(* PLC project benzene-distillation, Generated TextualNotationConverter 1.0 *)
(* stored: creationDateTime 2025-07-30T12:00:00, modificationDateTime 2025-01-30T12:00:00 *)

FUNCTION_BLOCK ANALOG_IN
  VAR_INPUT
    Name : STRING;
    Description : STRING;
    Raw_Signal : REAL;
    PV_High : REAL;
    PV_Low : REAL;
    Scaling_Slope : REAL;
    Scaling_Offset : REAL;
    Alarm_Enable : BOOL;
  END_VAR
  VAR_OUTPUT
    PV : REAL;
    High_Alarm : BOOL;
    Low_Alarm : BOOL;
    General_Fault : BOOL;
  END_VAR

            
          
END_FUNCTION_BLOCK

FUNCTION_BLOCK DIGITAL_IN
  VAR_INPUT
    Name : STRING;
    Description : STRING;
    DI_Raw : BOOL;
    DebounceTime : STRING;
    EnableAlarm : BOOL;
  END_VAR
  VAR_OUTPUT
    DI_Out : BOOL;
    Fault_State : BOOL;
  END_VAR

            
          
END_FUNCTION_BLOCK

FUNCTION_BLOCK PID_BASIC
  VAR_INPUT
    Name : STRING;
    Description : STRING;
    AUTO : BOOL;
    PV : REAL;
    SP : REAL;
    MV_MIN : REAL;
    MV_MAX : REAL;
    X0 : REAL;
    KP : REAL;
    TR : REAL;
    TD : REAL;
    PV_High : REAL;
    PV_Low : REAL;
    Deviation_Limit : REAL;
    Inhibit : BOOL;
  END_VAR
  VAR_OUTPUT
    PV_High_Alarm : BOOL;
    PV_Low_Alarm : BOOL;
    Deviation_Alarm : BOOL;
    XOUT : REAL;
  END_VAR

            
          
END_FUNCTION_BLOCK

FUNCTION_BLOCK VALVE_ELECTRIC
  VAR_INPUT
    Name : STRING;
    Description : STRING;
    Control_Signal : REAL;
    Manual_Mode : BOOL;
    Manual_Position : REAL;
    Open_Limit : REAL;
    Close_Limit : REAL;
    Timeout : STRING;
    Inhibit : BOOL;
  END_VAR
  VAR_OUTPUT
    Valve_Position : REAL;
    Feedback_Pos : REAL;
    Valve_Moving : BOOL;
    Position_Error : BOOL;
    Alarm : BOOL;
  END_VAR

            
          
END_FUNCTION_BLOCK

FUNCTION_BLOCK VALVE_ON_OFF
  VAR_INPUT
    Name : STRING;
    Description : STRING;
    Open_Cmd : BOOL;
    Close_Cmd : BOOL;
    Timeout : STRING;
    Inhibit : BOOL;
  END_VAR
  VAR_OUTPUT
    FB_Opened : BOOL;
    FB_Closed : BOOL;
    Valve_Open_Out : BOOL;
    Valve_Close_Out : BOOL;
    Alarm_Position_Error : BOOL;
    Alarm_General : BOOL;
  END_VAR

            
          
END_FUNCTION_BLOCK

PROGRAM Section2
  VAR
    TE101_BaseTemp_PV : REAL;
    PV103_MV_Command : REAL;
    PV103_Position_Feedback : REAL;
    XV105_Open_Feedback : BOOL;
    LIT101_ColumnLevel_PV : REAL;
    PIT102_Pressure_PV : REAL;
  END_VAR
  VAR
    TE-101 : ANALOG_IN;
    TIC-104 : PID_BASIC;
    PV-103 : VALVE_ELECTRIC;
    XV-105 : VALVE_ON_OFF;
    LIT-101 : ANALOG_IN;
    PIT-102 : ANALOG_IN;
    LAH-101 : DIGITAL_IN;
    LAL-101 : DIGITAL_IN;
  END_VAR
  VAR  (* added by the conversion: wires and edge detectors of the diagram *)
    _OR1_OUT : BOOL;
  END_VAR

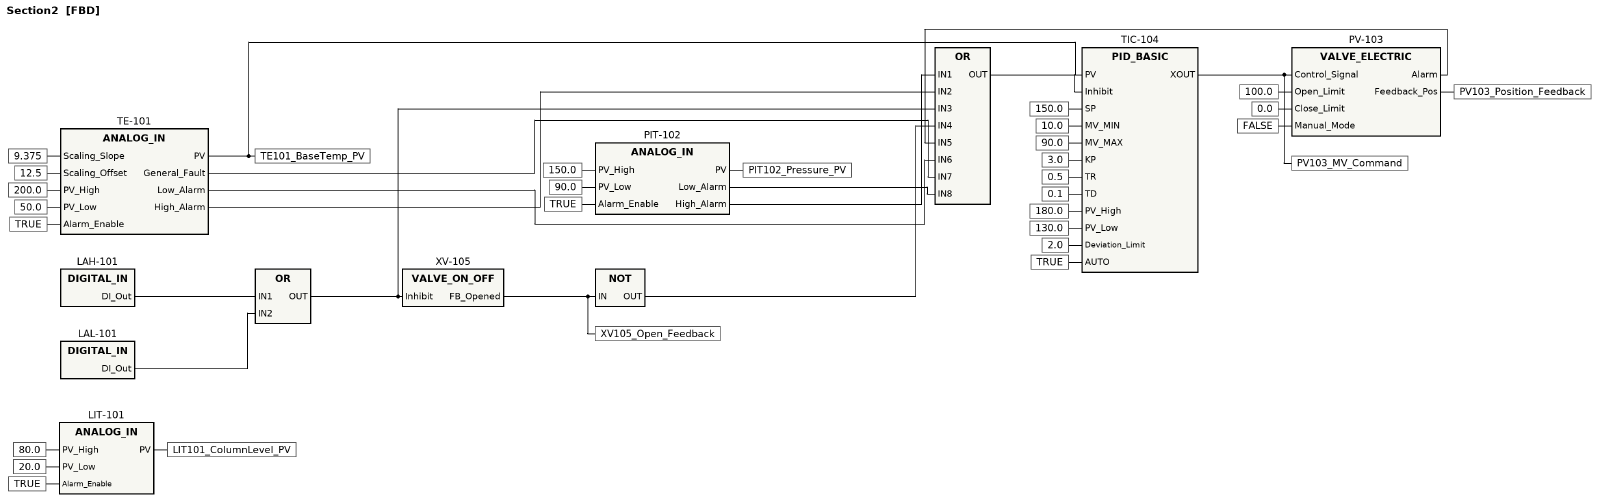
(* FBD diagram, written out as Structured Text *)
LIT-101(PV_High := 80.0, PV_Low := 20.0, Alarm_Enable := TRUE);
LIT101_ColumnLevel_PV := LIT-101.PV;
PIT-102(PV_High := 150.0, PV_Low := 90.0, Alarm_Enable := TRUE);
PIT102_Pressure_PV := PIT-102.PV;
TE-101(Scaling_Slope := 9.375, Scaling_Offset := 12.5, PV_High := 200.0, PV_Low := 50.0, Alarm_Enable := TRUE);
LAH-101();
LAL-101();
_OR1_OUT := LAH-101.DI_Out OR LAL-101.DI_Out;
XV-105(Inhibit := _OR1_OUT);
PV-103(Control_Signal := TIC-104.XOUT, Open_Limit := 100.0, Close_Limit := 0.0, Manual_Mode := FALSE);
TIC-104(PV := TE-101.PV, Inhibit := PIT-102.High_Alarm OR TE-101.High_Alarm OR _OR1_OUT OR NOT XV-105.FB_Opened OR PV-103.Alarm OR TE-101.Low_Alarm OR TE-101.General_Fault OR PIT-102.Low_Alarm, SP := 150.0, MV_MIN := 10.0, MV_MAX := 90.0, KP := 3.0, TR := 0.5, TD := 0.1, PV_High := 180.0, PV_Low := 130.0, Deviation_Limit := 2.0, AUTO := TRUE);
PV103_MV_Command := TIC-104.XOUT;
PV103_Position_Feedback := PV-103.Feedback_Pos;
TE101_BaseTemp_PV := TE-101.PV;
XV105_Open_Feedback := XV-105.FB_Opened;
END_PROGRAM

FUNCTION_BLOCK BOOL_IN
  VAR_INPUT
    Name : STRING;
    Description : STRING;
    Bool_In : BOOL;
    Alarm_OnTrue : BOOL;
    Alarm_OnFalse : BOOL;
    Latch_Enable : BOOL;
    Reset_Latch : BOOL;
  END_VAR
  VAR_OUTPUT
    Bool_Out : BOOL;
    Alarm_Active : BOOL;
    Latched_Status : BOOL;
  END_VAR

            
          
END_FUNCTION_BLOCK

FUNCTION_BLOCK DUTY_STANDBY
  VAR_INPUT
    Name : STRING;
    Description : STRING;
    Enable : BOOL;
    StartRequest : BOOL;
    AlternateEnable : BOOL;
    ForcePumpA : BOOL;
    ForcePumpB : BOOL;
    DutyElapsed : BOOL;
    MinRunElapsed : BOOL;
    SwitchoverDelayElapsed : BOOL;
    StartTimeoutElapsed : BOOL;
    PumpA_RunFB : BOOL;
    PumpB_RunFB : BOOL;
    PumpA_Fault : BOOL;
    PumpB_Fault : BOOL;
    Reset : BOOL;
    Inhibit : BOOL;
  END_VAR
  VAR_OUTPUT
    CmdPumpA : BOOL;
    CmdPumpB : BOOL;
    ActiveIsA : BOOL;
    SwitchedDueToDuty : BOOL;
    SwitchedDueToFailure : BOOL;
    Alarm_FailedStart_A : BOOL;
    Alarm_FailedStart_B : BOOL;
    Alarm_NoAvailablePump : BOOL;
  END_VAR

            
          
END_FUNCTION_BLOCK

FUNCTION_BLOCK MOTOR_2SPD
  VAR_INPUT
    Name : STRING;
    Description : STRING;
    Start_Cmd : BOOL;
    Stop_Cmd : BOOL;
    Speed_High_Cmd : BOOL;
    Speed_Low_Cmd : BOOL;
    Inhibit : BOOL;
  END_VAR
  VAR_OUTPUT
    Motor_Start_Out : BOOL;
    FB_Running : BOOL;
    FB_Trip : BOOL;
    FB_HighSpeed : BOOL;
    FB_LowSpeed : BOOL;
    Alarm_Speed_Error : BOOL;
  END_VAR

            
          
END_FUNCTION_BLOCK

FUNCTION_BLOCK MOTOR_ON_OFF
  VAR_INPUT
    Name : STRING;
    Description : STRING;
    Start_Cmd : BOOL;
    Stop_Cmd : BOOL;
    Start_Delay : STRING;
    MinRunTime : STRING;
    Inhibit : BOOL;
  END_VAR
  VAR_OUTPUT
    Motor_Start_Out : BOOL;
    FB_Running : BOOL;
    FB_Trip : BOOL;
    Alarm_Start_Fail : BOOL;
    Alarm_Stop_Fail : BOOL;
  END_VAR

            
          
END_FUNCTION_BLOCK

FUNCTION_BLOCK MOTOR_VSD
  VAR_INPUT
    Name : STRING;
    Description : STRING;
    Start_Cmd : BOOL;
    Stop_Cmd : BOOL;
    Speed_SP : REAL;
    Accel_Ramp : STRING;
    Decel_Ramp : STRING;
    Inhibit : BOOL;
  END_VAR
  VAR_OUTPUT
    Speed_Out : REAL;
    FB_Running : BOOL;
    FB_Fault : BOOL;
    FB_Ready : BOOL;
    FB_ActualSpeed : REAL;
    Alarm_Speed_Deviation : BOOL;
    Alarm_Comm_Fail : BOOL;
  END_VAR

            
          
END_FUNCTION_BLOCK

FUNCTION_BLOCK RATIO_CONTROL
  VAR_INPUT
    Name : STRING;
    Description : STRING;
    Auto : BOOL;
    PrimaryPV : REAL;
    SecondaryPV : REAL;
    RatioSP : REAL;
    Bias : REAL;
    TrimKp : REAL;
    TrimTi : STRING;
    MV_MIN : REAL;
    MV_MAX : REAL;
    ManOut : REAL;
    Inhibit : BOOL;
  END_VAR
  VAR_OUTPUT
    SlaveSP : REAL;
    ActiveRatio : REAL;
    RatioErr : REAL;
  END_VAR

            
          
END_FUNCTION_BLOCK

FUNCTION_BLOCK SPLIT_RANGE
  VAR_INPUT
    Name : STRING;
    Description : STRING;
    IN : REAL;
    Split_Point : REAL;
    Output1_Start : REAL;
    Output1_End : REAL;
    Output2_Start : REAL;
    Output2_End : REAL;
  END_VAR
  VAR_OUTPUT
    OUT1 : REAL;
    OUT2 : REAL;
  END_VAR

            
          
END_FUNCTION_BLOCK

FUNCTION_BLOCK VOTING_ANALOG
  VAR_INPUT
    Name : STRING;
    Description : STRING;
    Input1 : REAL;
    Input2 : REAL;
    Input3 : REAL;
    Deviation_Limit : REAL;
    Voting_Scheme : STRING;
    EnableAlarm : BOOL;
    Inhibit : BOOL;
  END_VAR
  VAR_OUTPUT
    Voted_Output : REAL;
    Sensor1_Fault : BOOL;
    Sensor2_Fault : BOOL;
    Sensor3_Fault : BOOL;
    Alarm_Voting_Error : BOOL;
    Healthy_Sensors_Count : INT;
  END_VAR

            
          
END_FUNCTION_BLOCK

PROGRAM Section3
  VAR
    TI_106_TemperaturePV : REAL;
    FIT_101_SteamFlowPV : REAL;
    PT_101_PressurePV : REAL;
    FIC_104_MV_Percent : REAL;
    LIC_002_LowLevelTrip : BOOL;
    FAH_104_FlowFailAlarm : BOOL;
    TAH_106_Alarm : BOOL;
    TAL_106_Alarm : BOOL;
    TCV_106_Alarm : BOOL;
    TCV_106_FeedbackPos : REAL;
  END_VAR
  VAR
    TI-106 : ANALOG_IN;
    FIT-101 : ANALOG_IN;
    PT-101 : ANALOG_IN;
    FIC-104 : PID_BASIC;
    TCV-106 : VALVE_ELECTRIC;
  END_VAR
  VAR  (* added by the conversion: wires and edge detectors of the diagram *)
    _OR42_OUT : BOOL;
  END_VAR

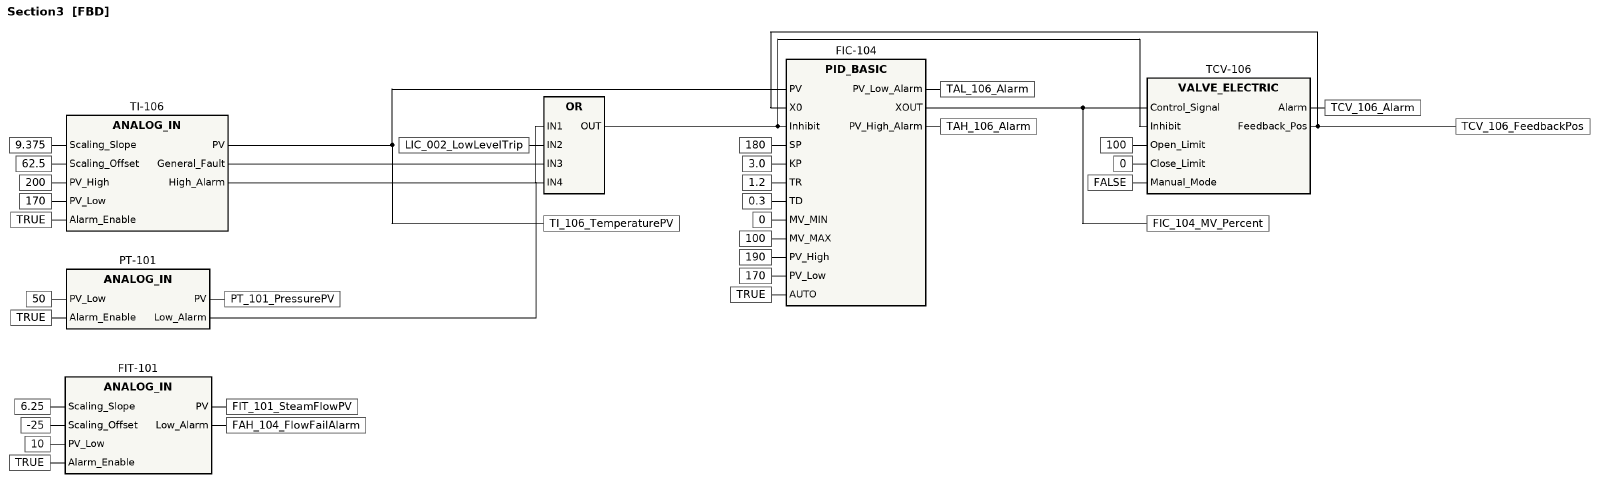
(* FBD diagram, written out as Structured Text *)
FIT-101(Scaling_Slope := 6.25, Scaling_Offset := -25, PV_Low := 10, Alarm_Enable := TRUE);
FAH_104_FlowFailAlarm := FIT-101.Low_Alarm;
TI-106(Scaling_Slope := 9.375, Scaling_Offset := 62.5, PV_High := 200, PV_Low := 170, Alarm_Enable := TRUE);
PT-101(PV_Low := 50, Alarm_Enable := TRUE);
_OR42_OUT := TI-106.High_Alarm OR LIC_002_LowLevelTrip OR TI-106.General_Fault OR PT-101.Low_Alarm;
TCV-106(Control_Signal := FIC-104.XOUT, Inhibit := _OR42_OUT, Open_Limit := 100, Close_Limit := 0, Manual_Mode := FALSE);
FIC-104(PV := TI-106.PV, X0 := TCV-106.Feedback_Pos, Inhibit := _OR42_OUT, SP := 180, KP := 3.0, TR := 1.2, TD := 0.3, MV_MIN := 0, MV_MAX := 100, PV_High := 190, PV_Low := 170, AUTO := TRUE);
FIC_104_MV_Percent := FIC-104.XOUT;
FIT_101_SteamFlowPV := FIT-101.PV;
PT_101_PressurePV := PT-101.PV;
TAH_106_Alarm := FIC-104.PV_High_Alarm;
TAL_106_Alarm := FIC-104.PV_Low_Alarm;
TCV_106_Alarm := TCV-106.Alarm;
TCV_106_FeedbackPos := TCV-106.Feedback_Pos;
TI_106_TemperaturePV := TI-106.PV;
END_PROGRAM

PROGRAM Section4
  VAR
    LT105_V104_Level_PV : REAL;
    FT107_CondensateFlow_PV : REAL;
    PT104_AccumulatorPressure_PV : REAL;
    LIC104_RSP_to_FIC107 : REAL;
    FIC107_ValveCmd_to_LV107 : REAL;
    XV103_Open_FB : BOOL;
    Cascade_Permissive_OK : BOOL;
    Startup_Delay_Done : BOOL;
  END_VAR
  VAR
    LT-105 : ANALOG_IN;
    FT-107 : ANALOG_IN;
    PT-104 : ANALOG_IN;
    LIC-104 : PID_BASIC;
    FIC-107 : PID_BASIC;
    PIC-104 : PID_BASIC;
    LV-107 : VALVE_ELECTRIC;
    XV-103 : VALVE_ON_OFF;
    LAH-104 : DIGITAL_IN;
    LAL-104 : DIGITAL_IN;
    StartupDelay : TON;
  END_VAR
  VAR  (* added by the conversion: wires and edge detectors of the diagram *)
    _OR83_OUT : BOOL;
    _NOT84_OUT : BOOL;
  END_VAR

(* FBD diagram, written out as Structured Text *)
PT-104(PV_High := 30.0, PV_Low := 15.0, Alarm_Enable := TRUE);
LT-105(PV_High := 90.0, PV_Low := 10.0, Alarm_Enable := TRUE);
XV-103();
FT-107(PV_Low := 0.0, PV_High := 50.0, Alarm_Enable := TRUE);
StartupDelay(IN := _NOT84_OUT, PT := T#30s);
LIC-104(PV := LT-105.PV, Inhibit := _OR83_OUT, AUTO := StartupDelay.Q, SP := 65.0, KP := 1.5, TR := 2.5, X0 := 40.0, MV_MIN := 0.0, MV_MAX := 100.0, PV_High := 90.0, PV_Low := 10.0);
FIC-107(SP := LIC-104.XOUT * 0.5, PV := FT-107.PV, Inhibit := _OR83_OUT, AUTO := _NOT84_OUT, KP := 4.0, TR := 0.5, MV_MIN := 0.0, MV_MAX := 100.0, X0 := 0.0);
LV-107(Control_Signal := FIC-107.XOUT, Inhibit := PT-104.High_Alarm, Manual_Mode := PT-104.High_Alarm, Manual_Position := 0.0, Close_Limit := 0.0, Open_Limit := 100.0);
_OR83_OUT := PT-104.High_Alarm OR PT-104.Low_Alarm OR LT-105.Low_Alarm OR NOT XV-103.FB_Opened OR FT-107.General_Fault OR LV-107.Position_Error;
_NOT84_OUT := NOT _OR83_OUT;
Cascade_Permissive_OK := _NOT84_OUT;
FIC107_ValveCmd_to_LV107 := FIC-107.XOUT;
FT107_CondensateFlow_PV := FT-107.PV;
LIC104_RSP_to_FIC107 := LIC-104.XOUT;
LT105_V104_Level_PV := LT-105.PV;
PT104_AccumulatorPressure_PV := PT-104.PV;
Startup_Delay_Done := StartupDelay.Q;
XV103_Open_FB := XV-103.FB_Opened;
PIC-104(PV := PT-104.PV, PV_High := 30.0, PV_Low := 15.0, MV_MIN := 0.0, MV_MAX := 100.0);
LAH-104();
LAL-104();
END_PROGRAM

PROGRAM Section5
  VAR
    FI102_FlowRate_PV : REAL;
    PI102_Pressure_PV : REAL;
    LIC102_Level_StartPermissive : BOOL;
    P102_ActiveIsA_Status : BOOL;
  END_VAR
  VAR
    FI-102 : ANALOG_IN;
    PI-102 : ANALOG_IN;
    LCV-102 : VALVE_ELECTRIC;
    LIC-102 : BOOL_IN;
    P-102A : MOTOR_ON_OFF;
    P-102B : MOTOR_ON_OFF;
    P-102 : DUTY_STANDBY;
  END_VAR
  VAR  (* added by the conversion: wires and edge detectors of the diagram *)
    _TON140_OUT : BOOL;
  END_VAR

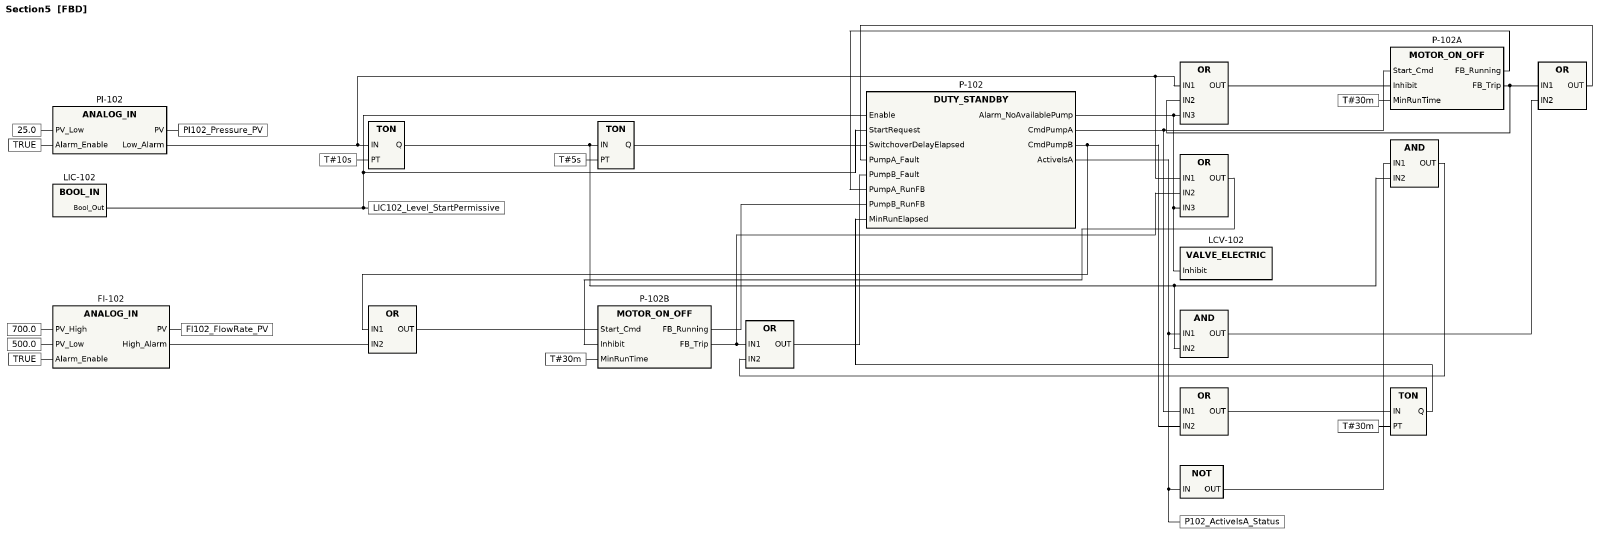
(* FBD diagram, written out as Structured Text *)
FI-102(PV_High := 700.0, PV_Low := 500.0, Alarm_Enable := TRUE);
FI102_FlowRate_PV := FI-102.PV;
LIC-102();
LIC102_Level_StartPermissive := LIC-102.Bool_Out;
PI-102(PV_Low := 25.0, Alarm_Enable := TRUE);
_TON140_OUT := TON(PI-102.Low_Alarm, T#10s);
P-102A(Start_Cmd := P-102.CmdPumpA, Inhibit := PI-102.Low_Alarm OR P-102A.FB_Trip OR P-102.Alarm_NoAvailablePump, MinRunTime := T#30m);
P-102B(Start_Cmd := P-102.CmdPumpB OR FI-102.High_Alarm, Inhibit := PI-102.Low_Alarm OR P-102B.FB_Trip OR P-102.Alarm_NoAvailablePump, MinRunTime := T#30m);
P-102(Enable := LIC-102.Bool_Out, StartRequest := LIC-102.Bool_Out, SwitchoverDelayElapsed := TON(_TON140_OUT, T#5s), PumpA_Fault := P-102A.FB_Trip OR P-102.ActiveIsA AND _TON140_OUT, PumpB_Fault := P-102B.FB_Trip OR NOT P-102.ActiveIsA AND _TON140_OUT, PumpA_RunFB := P-102A.FB_Running, PumpB_RunFB := P-102B.FB_Running, MinRunElapsed := TON(P-102.CmdPumpA OR P-102.CmdPumpB, T#30m));
P102_ActiveIsA_Status := P-102.ActiveIsA;
PI102_Pressure_PV := PI-102.PV;
LCV-102(Inhibit := P-102.Alarm_NoAvailablePump);
END_PROGRAM

PROGRAM Section6
  VAR
    FT105_FeedFlowRate : REAL;
    FT106_BottomsFlowRate : REAL;
    FT106_FlowSP_FromRatio : REAL;
  END_VAR
  VAR
    FT-105 : ANALOG_IN;
    FT-106 : ANALOG_IN;
    FV-101 : VALVE_ELECTRIC;
    IIC-104 : RATIO_CONTROL;
    FIC-106 : PID_BASIC;
    LIC-002 : PID_BASIC;
    FEED_PUMP_RUN : DIGITAL_IN;
    BOTTOMS_PUMP_RUN : DIGITAL_IN;
  END_VAR
  VAR  (* added by the conversion: wires and edge detectors of the diagram *)
    _OR171_OUT : BOOL;
  END_VAR

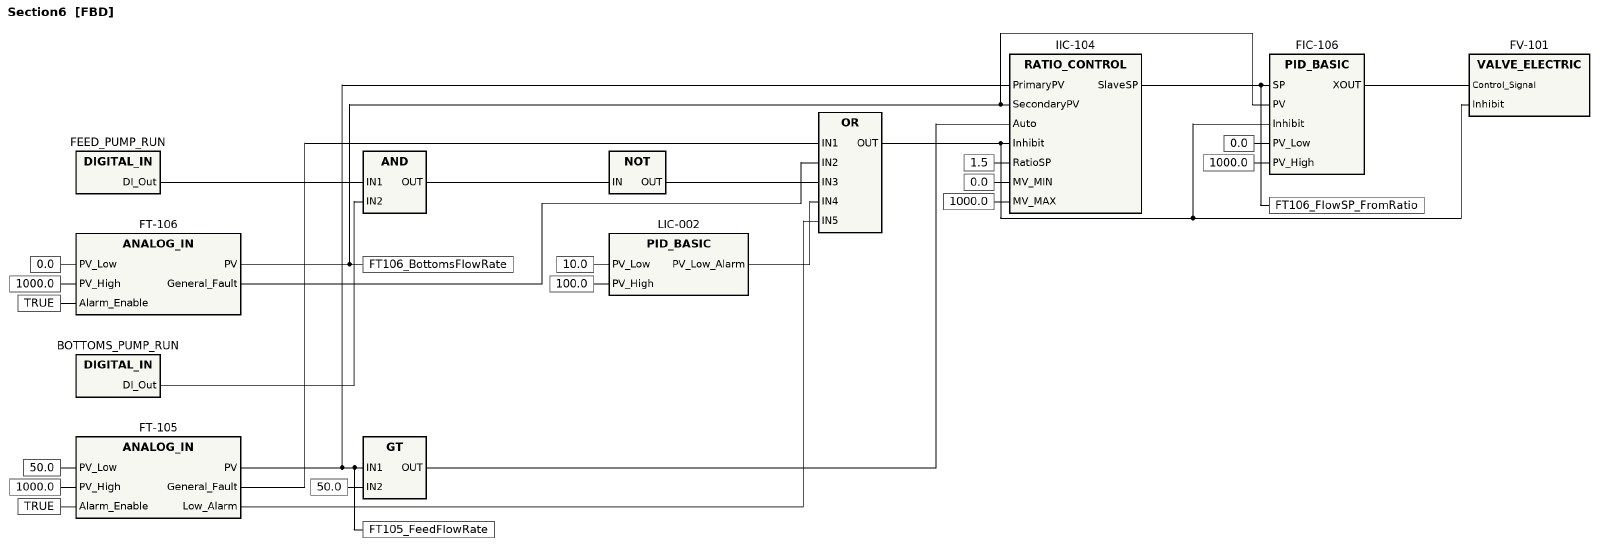
(* FBD diagram, written out as Structured Text *)
FT-105(PV_Low := 50.0, PV_High := 1000.0, Alarm_Enable := TRUE);
FT105_FeedFlowRate := FT-105.PV;
FT-106(PV_Low := 0.0, PV_High := 1000.0, Alarm_Enable := TRUE);
FT106_BottomsFlowRate := FT-106.PV;
FEED_PUMP_RUN();
BOTTOMS_PUMP_RUN();
LIC-002(PV_Low := 10.0, PV_High := 100.0);
_OR171_OUT := FT-105.General_Fault OR FT-106.General_Fault OR NOT (FEED_PUMP_RUN.DI_Out AND BOTTOMS_PUMP_RUN.DI_Out) OR LIC-002.PV_Low_Alarm OR FT-105.Low_Alarm;
IIC-104(PrimaryPV := FT-105.PV, SecondaryPV := FT-106.PV, Auto := FT-105.PV > 50.0, Inhibit := _OR171_OUT, RatioSP := 1.5, MV_MIN := 0.0, MV_MAX := 1000.0);
FT106_FlowSP_FromRatio := IIC-104.SlaveSP;
FIC-106(SP := IIC-104.SlaveSP, PV := FT-106.PV, Inhibit := _OR171_OUT, PV_Low := 0.0, PV_High := 1000.0);
FV-101(Control_Signal := FIC-106.XOUT, Inhibit := _OR171_OUT);
END_PROGRAM

CONFIGURATION Config0
  RESOURCE Res0 ON PLC
    TASK task0(INTERVAL := T#20ms, PRIORITY := 0);
    PROGRAM instance0 WITH task0 : Section2;
    PROGRAM instance_1 WITH task0 : Section3;
    PROGRAM instance_2 WITH task0 : Section4;
    PROGRAM instance_3 WITH task0 : Section5;
    PROGRAM instance_4 WITH task0 : Section6;
  END_RESOURCE
END_CONFIGURATION
